(* IEC 61131-3 sources: Shell-Scripting/, 8 files *)

(* ---- ADLFPT5.st ---- *)
DATA_BLOCK AutomatedDisassemblyLineDB
  VAR
    powerToolType: INT;
    components: ARRAY[1..N] OF COMPONENT;  (* Define a data structure for components *)
    inspectionPassed: BOOL;
    toolAvailable: BOOL;
  END_VAR
END_DATA_BLOCK

FUNCTION_BLOCK AutomatedDisassemblyLine
  METHODS
    IdentifyPowerTool : INT;
    DisassemblePowerTool : INT, components : ARRAY[1..N] OF COMPONENT;
    QualityInspection : components : ARRAY[1..N] OF COMPONENT;
    SortAndRecycle : components : ARRAY[1..N] OF COMPONENT;
    PowerToolAvailable : BOOL;
  END_METHODS

  METHODS IMPLEMENTATION
    IdentifyPowerTool : INT
      (* Implement vision system logic to identify the type of power tool *)
      RETURN powerToolType;
    END_METHOD

    DisassemblePowerTool : INT, components : ARRAY[1..N] OF COMPONENT
      (* Implement disassembly steps for the specific power tool type *)
      (* Example: remove screws, open casing, extract battery, etc. *)
    END_METHOD

    QualityInspection : components : ARRAY[1..N] OF COMPONENT
      (* Implement inspection logic for wear, damage, or defects *)
      (* Mark components as reusable or non-reusable *)
      RETURN inspectionPassed;
    END_METHOD

    SortAndRecycle : components : ARRAY[1..N] OF COMPONENT
      (* Implement sorting logic for recycling or further processing *)
      (* Example: separate reusable components from non-reusable ones *)
    END_METHOD

    PowerToolAvailable : BOOL
      (* Implement logic to check if there is a power tool available *)
      RETURN toolAvailable;
    END_METHOD
  END_METHODS
END_FUNCTION_BLOCK

(* ---- ADLFPT7.st ---- *)
FUNCTION_BLOCK DisassemblyLine
VAR_INPUT
    powerToolIn: BOOL; // Input signal indicating the presence of a power tool on the line
END_VAR

VAR_OUTPUT
    disassembled: BOOL; // Output signal indicating if the power tool has been disassembled
END_VAR

VAR
    conveyorRunning: BOOL := FALSE; // Internal variable to track the state of the conveyor
    disassemblyToolRunning: BOOL := FALSE; // Internal variable to track the state of the disassembly tool
END_VAR

METHOD DisassemblyProcess: BOOL
VAR
    powerToolDetected: BOOL := FALSE; // Internal variable to detect the presence of a power tool
    disassembledTool: BOOL := FALSE; // Internal variable to track the disassembly process
END_VAR

    // Check if a power tool is present on the line
    powerToolDetected := powerToolIn;

    IF powerToolDetected THEN
        // Start the conveyor
        conveyorRunning := TRUE;

        // Start the disassembly tool
        disassemblyToolRunning := TRUE;

        // Perform the disassembly process
        // ...

        // Set the output signal to indicate that the power tool has been disassembled
        disassembled := disassembledTool;
    ELSE
        // Stop the conveyor
        conveyorRunning := FALSE;

        // Stop the disassembly tool
        disassemblyToolRunning := FALSE;

        // Reset the output signal
        disassembled := FALSE;
    END_IF;

    // Return the status of the disassembly process
    RETURN disassembled;
END_METHOD

(* ---- ADLFPT_Final.st ---- *)
DATA_BLOCK AutomatedDisassemblyLineDB
  VAR
    powerToolAvailable: BOOL := FALSE; // Input signal indicating the presence of a power tool on the line.
    disassemblyInspectionPassed: BOOL := FALSE; // Output signal indicating the status of disassembly process.
    cellIndicator: INT := 0; // A constant variable for cell identifier.
    powerToolData: STRUCT;
    (* A data structure for power tool's physical informtion.
    The structure is output of pre-processing stage;
    i.e., information from load cell, position sensor, vision system, etc
    is collected and stored into this variable.*)
    disassemblyPerformanceData: STRUCT;
    (* A data structure for disassembly process informtion.
    The structure is output of quality inspection of disassembly process.
    The variable can be used as an indicator of damage or defect level,
    as well as a feedback for tuning and improving robot performance.*)
    sortedComponents: INT;
    (*Output variable indicating the status of disassembled components.
    The variable is the result of sorting process,
    and can be used as a measure for seprating cells from non-cells components.*)
    cellData: STRUCT;
    (* A data structure for battery cell's informtion.
    The structure is output of classification stage;
    i.e., information from cell inspection, cell life test, etc
    is collected and stored into this variable.*)
  END_VAR
END_DATA_BLOCK

FUNCTION_BLOCK AutomatedDisassemblyLine
  METHODS
    CheckPowerToolPresence : BOOL;
    IdentifyPowerTool : STRUCT;
    DisassemblePowerTool(powerToolData: STRUCT) : BOOL, STRUCT;
    SortComponents : INT;
    InspectCellSpecification: STRUCT;
  END_METHODS

  METHODS IMPLEMENTATION
    CheckPowerToolPresence : BOOL
      (* Implement logic to check if there is a power tool available.*)
      RETURN powerToolAvailable;
    END_METHOD

    IdentifyPowerTool : STRUCT
      (* Implement logic for pre-processing stage; i.e. collecting object's information.*)
      RETURN powerToolData;
    END_METHOD

    DisassemblePowerTool(powerToolData: STRUCT) : BOOL, STRUCT
      (* Implement disassembly steps such as removing screws, openning the casing, extract the battery modules, etc.*)
      (* The method is an interface between the proccessing unit and the robot.*)
      RETURN disassemblyInspectionPassed, disassemblyPerformanceData;
    END_METHOD

    SortComponents : INT
      (* Implement sorting logic in order to identify the components.*)
      RETURN  sortedComponents;
    END_METHOD

    InspectCellSpecification: STRUCT
      (* Implement classification logic for battery cells.*)
      RETURN cellData;
    END_METHOD
  END_METHODS

  (* Main program *)
  // Check if a power tool is present on the line.
  CheckPowerToolPresence();
  // Start the pre-processing stage.
  IF powerToolAvailable THEN
    IdentifyPowerTool();
  END_IF;
  // Perform the disassembly process.
  DisassemblePowerTool(powerToolData);
  IF disassemblyInspectionPassed THEN
    // Performing the sorting process.
    SortComponents();
  END_IF;
  IF sortedComponents = cellIndicator THEN
    // Perform cell classification
    InspectCellSpecification();
  END_IF;
END_FUNCTION_BLOCK

(* ---- ADLFPT_KUKA04.st ---- *)
(* Define a class for the power tool *)
CLASS PowerTool
  PRIVATE
    serialNumber : STRING;  (* Serial number of the power tool *)
    weight : REAL;  (* Weight of the power tool *)
    // Add other properties and methods as needed
  PUBLIC
    CONSTRUCTOR Init(serial: STRING, toolWeight: REAL)
      serialNumber := serial;
      weight := toolWeight;
    END_CONSTRUCTOR

    METHOD Disassemble()
      // Add code to disassemble the power tool
    END_METHOD
END_CLASS

(* Define a class for the disassembly line *)
CLASS DisassemblyLine
  PRIVATE
    robot : mxAutomation.ROBOT;  (* KUKA robot for disassembly *)
    conveyorBelt : ConveyorBelt;  (* Conveyor belt for transporting power tools *)
    // Add other components as needed
  PUBLIC
    CONSTRUCTOR Init(robotName: STRING)
      robot := mxAutomation.ROBOT.Create(robotName);
      // Initialize other components of the disassembly line
    END_CONSTRUCTOR

    METHOD StartDisassemblyLine()
      // Add code to start the disassembly line
      // Activate conveyor belt, initialize robot, etc.
    END_METHOD

    METHOD StopDisassemblyLine()
      // Add code to stop the disassembly line
      // Deactivate conveyor belt, shut down robot, etc.
    END_METHOD

    METHOD DisassemblePowerTool(tool: PowerTool)
      // Call the Disassemble method of the PowerTool object
      tool.Disassemble();
    END_METHOD
END_CLASS

(* Main program *)
PROGRAM MainProgram
VAR
  disassemblyLine : DisassemblyLine;  (* Disassembly line object *)
  powerTool1 : PowerTool;  (* First power tool object *)
  powerTool2 : PowerTool;  (* Second power tool object *)
END_VAR

(* Initialize the disassembly line with the KUKA robot *)
disassemblyLine := DisassemblyLine.Init("Robot1");

(* Create instances of power tools with serial numbers and weights *)
powerTool1 := PowerTool.Init("SN123", 5.0);
powerTool2 := PowerTool.Init("SN456", 6.0);

(* Start the disassembly line and disassemble the power tools *)
disassemblyLine.StartDisassemblyLine();
disassemblyLine.DisassemblePowerTool(powerTool1);
disassemblyLine.DisassemblePowerTool(powerTool2);
disassemblyLine.StopDisassemblyLine();

END_PROGRAM

(* ---- ADLFPT4.st ---- *)
PROGRAM AutomatedDisassemblyLine
VAR
  powerToolType: INT;
  components: ARRAY[1..N] OF COMPONENT;  (* Define a data structure for components *)

FUNCTION IdentifyPowerTool: INT
  (* Use vision system to identify the type of power tool *)
  RETURN powerToolType;
END_FUNCTION;

FUNCTION DisassemblePowerTool(toolType: INT)
  (* Perform disassembly steps for the specific power tool type *)
  (* Example: remove screws, open casing, extract battery, etc. *)
  (* Implement robot movements and actions *)
END_FUNCTION;

FUNCTION QualityInspection(components: ARRAY): BOOL
  (* Inspect disassembled components for wear, damage, or defects *)
  (* Mark components as reusable or non-reusable *)
  RETURN inspectionPassed;
END_FUNCTION;

FUNCTION SortAndRecycle(components: ARRAY)
  (* Sort components for recycling or further processing *)
  (* Example: separate reusable components from non-reusable ones *)
  (* Implement sorting mechanism *)
END_FUNCTION;

FUNCTION PowerToolAvailable: BOOL
  (* Check if there is a power tool available on the disassembly line *)
  RETURN toolAvailable;
END_FUNCTION;

VAR
  inspectionPassed: BOOL;
  toolAvailable: BOOL;

(* Main program *)
AUTOMATED_DISASSEMBLY_LINE:
  REPEAT
    IF PowerToolAvailable() THEN
      powerToolType := IdentifyPowerTool();
      DisassemblePowerTool(powerToolType);
      inspectionPassed := QualityInspection(components);

      IF inspectionPassed THEN
        SortAndRecycle(components);
      END_IF;
    END_IF;
  END_REPEAT;
END_PROGRAM.

(* ---- ADLFPT_KUKA02.st ---- *)
PROGRAM MainProgram
VAR
    kukaRobot : mxAutomation.ROBOT;  (* Declare the KUKA robot variable *)
END_VAR

METHOD MoveRobotToStartingPosition : BOOL
VAR_INPUT
    startingPositionX : REAL;  (* X-coordinate of the starting position *)
    startingPositionY : REAL;  (* Y-coordinate of the starting position *)
    startingPositionZ : REAL;  (* Z-coordinate of the starting position *)
END_VAR
VAR
    success : BOOL;  (* Variable to store the success status of the movement *)
END_VAR

(* Initialize the mxAutomation package and connect to the robot *)
kukaRobot := mxAutomation.ROBOT.Create("RobotName");  (* Replace "RobotName" with the actual name of the robot *)

(* Move the robot to the starting position *)
success := kukaRobot.MoveTo(startingPositionX, startingPositionY, startingPositionZ);

IF NOT success THEN
    (* Handle the case when the movement fails *)
    // Add your error handling code here
END_IF

END_METHOD

(* ---- ADLFPT_KUKA03.st ---- *)
PROGRAM MainProgram
VAR
    kukaRobot : mxAutomation.ROBOT;  (* Declare the KUKA robot variable *)
END_VAR

METHOD MoveRobotToStartingPosition : BOOL
VAR_INPUT
    startingPositionX : REAL;  (* X-coordinate of the starting position *)
    startingPositionY : REAL;  (* Y-coordinate of the starting position *)
    startingPositionZ : REAL;  (* Z-coordinate of the starting position *)
END_VAR
VAR
    success : BOOL;  (* Variable to store the success status of the movement *)
END_VAR

(* Initialize the mxAutomation package and connect to the robot *)
kukaRobot := mxAutomation.ROBOT.Create("RobotName");  (* Replace "RobotName" with the actual name of the robot *)

(* Move the robot to the starting position using KRC_MoveLinearAbsolute *)
success := kukaRobot.KRC_MoveLinearAbsolute(startingPositionX, startingPositionY, startingPositionZ);

IF NOT success THEN
    (* Handle the case when the movement fails *)
    // Add your error handling code here
END_IF

END_METHOD

(* ---- ADLFPT_Robot.st ---- *)
VAR
    robotPosition: AXIS := 0;   (* Variable to store robot arm position *)
    toolInHand: BOOL := FALSE;  (* Variable to track whether the tool is in the robot's hand *)

METHOD RobotControl
    IF NOT toolInHand THEN
        MoveRobotToStartPosition();  (* Move the robot to the starting position *)
        toolInHand := PickUpTool();  (* Pick up the tool and update the status *)
    END_IF;

    ExecuteDisassemblyProcess();  (* Execute the disassembly process *)

    IF toolInHand THEN
        toolInHand := PlaceTool();  (* Place the tool and update the status *)
    END_IF;

    MoveRobotToNextPosition();  (* Move the robot to the next position for the next cycle *)
END_METHOD

METHOD MoveRobotToStartPosition
    (* Code to move the robot to the starting position *)
END_METHOD

METHOD PickUpTool : BOOL
    (* Code to control the robot to pick up the tool *)
    RETURN TRUE;  (* Return TRUE to indicate the tool is now in the robot's hand *)
END_METHOD

METHOD ExecuteDisassemblyProcess
    (* Code to control the robot to perform the disassembly process *)
END_METHOD

METHOD PlaceTool : BOOL
    (* Code to control the robot to place the tool *)
    RETURN FALSE;  (* Return FALSE to indicate the tool is no longer in the robot's hand *)
END_METHOD

METHOD MoveRobotToNextPosition
    (* Code to move the robot to the next position for the next cycle *)
END_METHOD
